Universal Robots PolyScope program: asm_idler_pulley_v1.urp

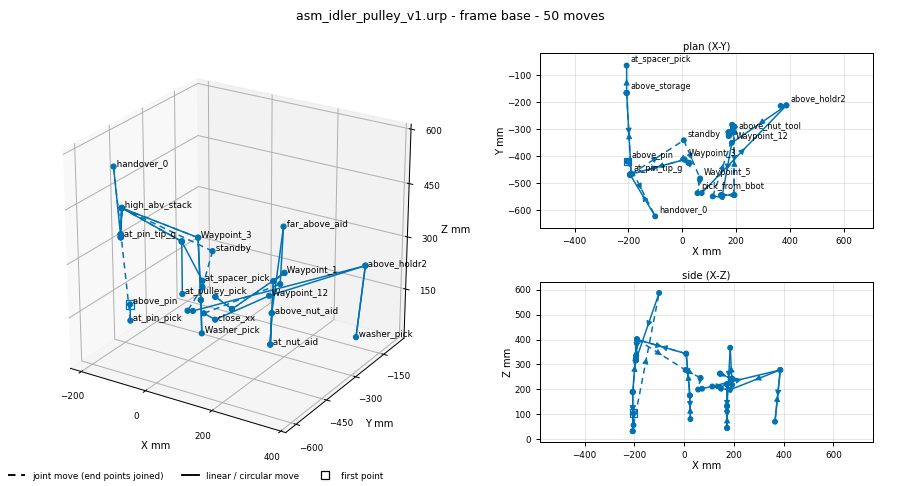
[picture p0: tool path of asm_idler_pulley_v1.urp in frame base, 50 of 58 moves have a stored position in this frame; points joined in program order, loops and branches not executed]
Program asm_idler_pulley_v1 (installation=default directory=/programs/wrs2020 createdIn=5.6.0.90886 lastSavedIn=5.9.1.1031110 robotSerialNumber=20205500180)
Calibrated DH parameters: a=[0, -0.425, -0.3922, 0, 0, 0]; d=[0.1625, 0, 0, 0.1333, 0.0997, 0.0996]; alpha=[1.570796, 0, 0, 1.570796, -1.570796, 0]; deltaTheta=[0, 0, 0, 0, 0, 0]
Robot Program (runOnlyOnce=true)
  var_1 := get_actual_joint_positions()
  MoveJ speed 60 deg/s, acceleration 80 deg/s^2 (useActiveTCP=true) feature=Base
    Waypoint Waypoint (Variable): variable=var_1
  URCap Gripper (Robotiq_Grippers, Robotiq Inc.) dataModel(position=70.98039215686275, force=100.0, speed=0.0, positionInDouble=70.98039215686275, forceInDouble=100.0, speedInDouble=0.0, slaveIds=[9], blocking=true)
  MoveL speed 50 mm/s, acceleration 1200 mm/s^2 (useActiveTCP=true) feature=Base
    Waypoint above_pin: motionParameters(jointSpeed=1.047198 jointAcceleration=1.396263 cartesianSpeed=0.5 cartesianAcceleration=1.2); TCP in base x=-203.451 y=-419.874 z=103.99 mm, rx=-2.2531 ry=-2.1572 rz=0.0025 rad; joints [48.461, -90.908, 115.612, -114.69, -91.283, 50.953] deg; TCP offset x=0 y=0 z=220 mm, rx=0 ry=0 rz=0 rad
    Waypoint at_pin_pick: motionParameters(jointSpeed=1.047198 jointAcceleration=1.396263 cartesianSpeed=0.5 cartesianAcceleration=1.2); TCP in base x=-203.465 y=-419.863 z=56.339 mm, rx=-2.2531 ry=-2.1571 rz=0.0025 rad; joints [48.46, -87.426, 120.005, -122.565, -91.284, 50.955] deg
  URCap Gripper (Robotiq_Grippers, Robotiq Inc.) dataModel(position=100.0, force=0.0, speed=0.0, positionInDouble=100.0, forceInDouble=0.0, speedInDouble=0.0, slaveIds=[9], blocking=true)
  MoveJ speed 60 deg/s, acceleration 80 deg/s^2 (useActiveTCP=true) feature=Base
    Waypoint handover_0: TCP in base x=-100.562 y=-623.369 z=587.469 mm, rx=1.5572 ry=0.0059 rz=0.0177 rad; joints [46.387, -101.66, 115.722, -195.155, -45.533, 181.192] deg
  Popup Message (haltProgram=false message=wait for b_bot to grasp pin. Press continue to release and proceed inputType=Text)
  URCap Gripper (Robotiq_Grippers, Robotiq Inc.) dataModel(position=34.90196078431372, force=100.0, speed=100.0, positionInDouble=34.90196078431372, forceInDouble=100.0, speedInDouble=100.0, slaveIds=[9], blocking=true)
  MoveL speed 250 mm/s, acceleration 1200 mm/s^2 (useActiveTCP=true) feature=Base
    MoveDirectionNode (selectedDirection=YPlus)
      Until DISTANCE (allowActions=false deceleration=3 distanceNodeType=STOP) Distance=0.08; motionParameters(blendRadius=0)
  Popup Message (haltProgram=false message=c when bbot moved down inputType=Text)
  Folder center pin
    MoveL speed 250 mm/s, acceleration 1200 mm/s^2 (useActiveTCP=true) feature=Base
      SuppressedNode
        Waypoint Waypoint_9: 
      Waypoint at_pin_tip_g: TCP in base x=-193.591 y=-468.719 z=318.204 mm, rx=3.1358 ry=0.014 rz=0.0168 rad; joints [51.873, -89.96, 82.562, -82.478, -89.318, 141.361] deg
    URCap Gripper (Robotiq_Grippers, Robotiq Inc.) dataModel(position=100.0, force=100.0, speed=100.0, positionInDouble=100.0, forceInDouble=100.0, speedInDouble=100.0, slaveIds=[9], blocking=true)
    URCap Gripper (Robotiq_Grippers, Robotiq Inc.) dataModel(position=41.96078431372549, force=100.0, speed=100.0, positionInDouble=41.96078431372549, forceInDouble=100.0, speedInDouble=100.0, slaveIds=[9], blocking=true)
    MoveL speed 800 mm/s, acceleration 1200 mm/s^2 (useActiveTCP=true) feature=Base
      Waypoint turn_left (Relative): relativeFromPosition TCP in base x=-247.487 y=-411.573 z=65.314 mm, rx=-0.0034 ry=-3.1246 rz=-0.0244 rad; joints [43.776, -86.347, 117.339, -121.073, -91.317, -46.099] deg; TCP in base x=-247.45 y=-411.548 z=65.274 mm, rx=2.2244 ry=-2.2172 rz=-0.0361 rad; joints [43.776, -86.344, 117.339, -121.066, -91.315, -136.41] deg
    URCap Gripper (Robotiq_Grippers, Robotiq Inc.) dataModel(position=100.0, force=100.0, speed=100.0, positionInDouble=100.0, forceInDouble=100.0, speedInDouble=100.0, slaveIds=[9], blocking=true)
    URCap Gripper (Robotiq_Grippers, Robotiq Inc.) dataModel(position=57.64705882352941, force=0.0, speed=0.0, positionInDouble=57.64705882352941, forceInDouble=0.0, speedInDouble=0.0, slaveIds=[9], blocking=true)
    MoveL speed 800 mm/s, acceleration 1200 mm/s^2 (useActiveTCP=true) feature=Base
      Waypoint turn_right (Relative): relativeFromPosition TCP in base x=-247.464 y=-411.551 z=65.306 mm, rx=2.2244 ry=-2.2171 rz=-0.0361 rad; joints [43.776, -86.348, 117.34, -121.068, -91.317, -136.413] deg; TCP in base x=-247.474 y=-411.554 z=65.268 mm, rx=-0.0035 ry=-3.1247 rz=-0.0244 rad; joints [43.774, -86.343, 117.34, -121.072, -91.315, -46.098] deg
    URCap Gripper (Robotiq_Grippers, Robotiq Inc.) dataModel(position=100.0, force=100.0, speed=100.0, positionInDouble=100.0, forceInDouble=100.0, speedInDouble=100.0, slaveIds=[9], blocking=true)
    URCap Gripper (Robotiq_Grippers, Robotiq Inc.) dataModel(position=0.0, force=100.0, speed=100.0, positionInDouble=0.0, forceInDouble=100.0, speedInDouble=100.0, slaveIds=[9], blocking=true)
  Folder get pulley
    MoveL speed 300 mm/s, acceleration 1200 mm/s^2 (useActiveTCP=true) feature=Base
      Waypoint above_storage: motionParameters(jointSpeed=1.047198 jointAcceleration=1.396263 cartesianSpeed=0.5 cartesianAcceleration=1.2 blendRadius=0.05); TCP in base x=-206.583 y=-165.263 z=189.567 mm, rx=3.1359 ry=0.0138 rz=0.017 rad; joints [7.844, -127.94, 126.119, -87.608, -89.601, 97.337] deg
      Waypoint at_pulley_pick: motionParameters(jointSpeed=1.047198 jointAcceleration=1.396263 cartesianSpeed=0.5 cartesianAcceleration=1.2); TCP in base x=-206.616 y=-165.272 z=31.944 mm, rx=3.1359 ry=0.0138 rz=0.0169 rad; joints [7.841, -121.393, 147.531, -115.569, -89.599, 97.336] deg
    Folder center+grasp
      URCap Gripper (Robotiq_Grippers, Robotiq Inc.) dataModel(position=100.0, force=0.0, speed=0.0, positionInDouble=100.0, forceInDouble=0.0, speedInDouble=0.0, slaveIds=[9], blocking=true)
      URCap Gripper (Robotiq_Grippers, Robotiq Inc.) dataModel(position=45.09803921568627, force=0.0, speed=0.0, positionInDouble=45.09803921568627, forceInDouble=0.0, speedInDouble=0.0, slaveIds=[9], blocking=true)
      MoveL speed 800 mm/s, acceleration 1200 mm/s^2 (useActiveTCP=true) feature=Base
        Waypoint turn_left (Relative): relativeFromPosition TCP in base x=-247.487 y=-411.573 z=65.314 mm, rx=-0.0034 ry=-3.1246 rz=-0.0244 rad; joints [43.776, -86.347, 117.339, -121.073, -91.317, -46.099] deg; TCP in base x=-247.45 y=-411.548 z=65.274 mm, rx=2.2244 ry=-2.2172 rz=-0.0361 rad; joints [43.776, -86.344, 117.339, -121.066, -91.315, -136.41] deg
      URCap Gripper (Robotiq_Grippers, Robotiq Inc.) dataModel(position=100.0, force=0.0, speed=0.0, positionInDouble=100.0, forceInDouble=0.0, speedInDouble=0.0, slaveIds=[9], blocking=true)
      URCap Gripper (Robotiq_Grippers, Robotiq Inc.) dataModel(position=57.64705882352941, force=0.0, speed=0.0, positionInDouble=57.64705882352941, forceInDouble=0.0, speedInDouble=0.0, slaveIds=[9], blocking=true)
      MoveL speed 800 mm/s, acceleration 1200 mm/s^2 (useActiveTCP=true) feature=Base
        Waypoint turn_right (Relative): relativeFromPosition TCP in base x=-247.464 y=-411.551 z=65.306 mm, rx=2.2244 ry=-2.2171 rz=-0.0361 rad; joints [43.776, -86.348, 117.34, -121.068, -91.317, -136.413] deg; TCP in base x=-247.474 y=-411.554 z=65.268 mm, rx=-0.0035 ry=-3.1247 rz=-0.0244 rad; joints [43.774, -86.343, 117.34, -121.072, -91.315, -46.098] deg
      URCap Gripper (Robotiq_Grippers, Robotiq Inc.) dataModel(position=100.0, force=0.0, speed=0.0, positionInDouble=100.0, forceInDouble=0.0, speedInDouble=0.0, slaveIds=[9], blocking=true)
  Folder stack pulley
    MoveJ speed 60 deg/s, acceleration 80 deg/s^2 (useActiveTCP=true) feature=Base
      Waypoint high_abv_stack: TCP in base x=-189.725 y=-466.715 z=400.408 mm, rx=3.1358 ry=0.0139 rz=0.0168 rad; joints [52.084, -87.731, 67.903, -70.048, -89.314, 141.575] deg
    MoveL speed 250 mm/s, acceleration 1200 mm/s^2 (useActiveTCP=true) feature=Base
      Waypoint at_tip_1: TCP in base x=-193.581 y=-468.753 z=326.241 mm, rx=3.1357 ry=0.014 rz=0.0167 rad; joints [51.875, -89.809, 81.226, -81.299, -89.316, 141.361] deg
    Folder push_down
      p_start := get_actual_tcp_pose()
      Force Frame feature=Base; selection=[0, 0, 1, 0, 0, 0]; wrench=[-5, 0, -5, 0, 0, 0]; limitsForce=[0.005, 0.15, 0.01, 1.047198, 1.047198, 1.047198]; limitsMotion=[0.1, 0.1, 0.1, 0.349066, 0.349066, 0.349066]
        MoveL speed 5 mm/s, acceleration 5 mm/s^2 (useActiveTCP=true) feature=Base
          Loop Counting (count=1) loopVariable(name=Loop_6)
            MoveDirectionNode (selectedDirection=YPlus) feature=Base
              Until DISTANCE (allowActions=false deceleration=3 distanceNodeType=STOP) Distance=0.001; motionParameters(blendRadius=0)
            MoveDirectionNode (selectedDirection=XPlus) feature=Base
              Until DISTANCE (allowActions=false deceleration=3 distanceNodeType=STOP) Distance=0.001; motionParameters(blendRadius=0)
            MoveDirectionNode (selectedDirection=YMinus) feature=Base
              Until DISTANCE (allowActions=false deceleration=3 distanceNodeType=STOP) Distance=0.001; motionParameters(blendRadius=0)
            MoveDirectionNode (selectedDirection=YMinus) feature=Base
              Until DISTANCE (allowActions=false deceleration=3 distanceNodeType=STOP) Distance=0.001; motionParameters(blendRadius=0)
            MoveDirectionNode (selectedDirection=XMinus) feature=Base
              Until DISTANCE (allowActions=false deceleration=3 distanceNodeType=STOP) Distance=0.001; motionParameters(blendRadius=0)
            MoveDirectionNode (selectedDirection=YPlus) feature=Base
              Until DISTANCE (allowActions=false deceleration=3 distanceNodeType=STOP) Distance=0.001; motionParameters(blendRadius=0)
            MoveDirectionNode (selectedDirection=YPlus) feature=Base
              Until DISTANCE (allowActions=false deceleration=3 distanceNodeType=STOP) Distance=0.001; motionParameters(blendRadius=0)
            MoveDirectionNode (selectedDirection=XMinus) feature=Base
              Until DISTANCE (allowActions=false deceleration=3 distanceNodeType=STOP) Distance=0.001; motionParameters(blendRadius=0)
            MoveDirectionNode (selectedDirection=YMinus) feature=Base
              Until DISTANCE (allowActions=false deceleration=3 distanceNodeType=STOP) Distance=0.001; motionParameters(blendRadius=0)
            MoveDirectionNode (selectedDirection=YMinus) feature=Base
              Until DISTANCE (allowActions=false deceleration=3 distanceNodeType=STOP) Distance=0.001; motionParameters(blendRadius=0)
            MoveDirectionNode (selectedDirection=XMinus) feature=Base
              Until DISTANCE (allowActions=false deceleration=3 distanceNodeType=STOP) Distance=0.001; motionParameters(blendRadius=0)
            MoveDirectionNode (selectedDirection=YPlus) feature=Base
              Until DISTANCE (allowActions=false deceleration=3 distanceNodeType=STOP) Distance=0.001; motionParameters(blendRadius=0)
        SuppressedNode
          Wait Sleep waitTime=4
      p_now := get_actual_tcp_pose()
      d := pose_dist(p_start,p_now)
      Popup Message (haltProgram=false inputType=Variable) variable=d
      If d < 0.01
        Popup Message (haltProgram=false message=fail? inputType=Text)
    URCap Gripper (Robotiq_Grippers, Robotiq Inc.) dataModel(position=41.96078431372549, force=100.0, speed=100.0, positionInDouble=41.96078431372549, forceInDouble=100.0, speedInDouble=100.0, slaveIds=[9], blocking=true)
    Folder recenter pin
      MoveL speed 250 mm/s, acceleration 1200 mm/s^2 (useActiveTCP=true) feature=Base
        Waypoint at_pin_tip_g: TCP in base x=-193.591 y=-468.719 z=318.204 mm, rx=3.1358 ry=0.014 rz=0.0168 rad; joints [51.873, -89.96, 82.562, -82.478, -89.318, 141.361] deg
      URCap Gripper (Robotiq_Grippers, Robotiq Inc.) dataModel(position=100.0, force=100.0, speed=100.0, positionInDouble=100.0, forceInDouble=100.0, speedInDouble=100.0, slaveIds=[9], blocking=true)
      URCap Gripper (Robotiq_Grippers, Robotiq Inc.) dataModel(position=41.96078431372549, force=100.0, speed=100.0, positionInDouble=41.96078431372549, forceInDouble=100.0, speedInDouble=100.0, slaveIds=[9], blocking=true)
    MoveJ speed 60 deg/s, acceleration 80 deg/s^2 (useActiveTCP=true) feature=Base
      Waypoint high_abv_stack: TCP in base x=-189.725 y=-466.715 z=400.408 mm, rx=3.1358 ry=0.0139 rz=0.0168 rad; joints [52.084, -87.731, 67.903, -70.048, -89.314, 141.575] deg
  Folder get spacer
    MoveL speed 300 mm/s, acceleration 1200 mm/s^2 (useActiveTCP=true) feature=Base
      Waypoint above_storage: motionParameters(jointSpeed=1.047198 jointAcceleration=1.396263 cartesianSpeed=0.5 cartesianAcceleration=1.2 blendRadius=0.05); TCP in base x=-206.583 y=-165.263 z=189.567 mm, rx=3.1359 ry=0.0138 rz=0.017 rad; joints [7.844, -127.94, 126.119, -87.608, -89.601, 97.337] deg
      Waypoint at_spacer_pick: motionParameters(jointSpeed=1.047198 jointAcceleration=1.396263 cartesianSpeed=0.5 cartesianAcceleration=1.2); TCP in base x=-206.636 y=-63.72 z=31.971 mm, rx=3.1359 ry=0.0138 rz=0.0168 rad; joints [-21.062, -135.483, 151.426, -105.257, -89.924, 68.434] deg
    Folder center+grasp
      URCap Gripper (Robotiq_Grippers, Robotiq Inc.) dataModel(position=100.0, force=0.0, speed=0.0, positionInDouble=100.0, forceInDouble=0.0, speedInDouble=0.0, slaveIds=[9], blocking=true)
      URCap Gripper (Robotiq_Grippers, Robotiq Inc.) dataModel(position=61.96078431372549, force=100.0, speed=0.0, positionInDouble=61.96078431372549, forceInDouble=100.0, speedInDouble=0.0, slaveIds=[9], blocking=true)
      MoveL speed 800 mm/s, acceleration 1200 mm/s^2 (useActiveTCP=true) feature=Base
        Waypoint turn_left (Relative): relativeFromPosition TCP in base x=-247.487 y=-411.573 z=65.314 mm, rx=-0.0034 ry=-3.1246 rz=-0.0244 rad; joints [43.776, -86.347, 117.339, -121.073, -91.317, -46.099] deg; TCP in base x=-247.45 y=-411.548 z=65.274 mm, rx=2.2244 ry=-2.2172 rz=-0.0361 rad; joints [43.776, -86.344, 117.339, -121.066, -91.315, -136.41] deg
      URCap Gripper (Robotiq_Grippers, Robotiq Inc.) dataModel(position=100.0, force=0.0, speed=0.0, positionInDouble=100.0, forceInDouble=0.0, speedInDouble=0.0, slaveIds=[9], blocking=true)
      URCap Gripper (Robotiq_Grippers, Robotiq Inc.) dataModel(position=57.64705882352941, force=0.0, speed=0.0, positionInDouble=57.64705882352941, forceInDouble=0.0, speedInDouble=0.0, slaveIds=[9], blocking=true)
      MoveL speed 800 mm/s, acceleration 1200 mm/s^2 (useActiveTCP=true) feature=Base
        Waypoint turn_right (Relative): relativeFromPosition TCP in base x=-247.464 y=-411.551 z=65.306 mm, rx=2.2244 ry=-2.2171 rz=-0.0361 rad; joints [43.776, -86.348, 117.34, -121.068, -91.317, -136.413] deg; TCP in base x=-247.474 y=-411.554 z=65.268 mm, rx=-0.0035 ry=-3.1247 rz=-0.0244 rad; joints [43.774, -86.343, 117.34, -121.072, -91.315, -46.098] deg
      URCap Gripper (Robotiq_Grippers, Robotiq Inc.) dataModel(position=100.0, force=0.0, speed=0.0, positionInDouble=100.0, forceInDouble=0.0, speedInDouble=0.0, slaveIds=[9], blocking=true)
    MoveL speed 300 mm/s, acceleration 1200 mm/s^2 (useActiveTCP=true) feature=Base
      Waypoint above_storage: motionParameters(jointSpeed=1.047198 jointAcceleration=1.396263 cartesianSpeed=0.5 cartesianAcceleration=1.2); TCP in base x=-206.583 y=-165.263 z=189.567 mm, rx=3.1359 ry=0.0138 rz=0.017 rad; joints [7.844, -127.94, 126.119, -87.608, -89.601, 97.337] deg
  Folder stack spacer
    MoveJ speed 60 deg/s, acceleration 80 deg/s^2 (useActiveTCP=true) feature=Base
      Waypoint high_abv_stack: TCP in base x=-189.725 y=-466.715 z=400.408 mm, rx=3.1358 ry=0.0139 rz=0.0168 rad; joints [52.084, -87.731, 67.903, -70.048, -89.314, 141.575] deg
    MoveL speed 250 mm/s, acceleration 1200 mm/s^2 (useActiveTCP=true) feature=Base
      Waypoint at_tip_1: TCP in base x=-193.581 y=-468.753 z=326.241 mm, rx=3.1357 ry=0.014 rz=0.0167 rad; joints [51.875, -89.809, 81.226, -81.299, -89.316, 141.361] deg
    Folder push_down
      p_start := get_actual_tcp_pose()
      Force Frame feature=Base; selection=[0, 0, 1, 0, 0, 0]; wrench=[-5, 0, -5, 0, 0, 0]; limitsForce=[0.005, 0.15, 0.01, 1.047198, 1.047198, 1.047198]; limitsMotion=[0.1, 0.1, 0.1, 0.349066, 0.349066, 0.349066]
        MoveL speed 5 mm/s, acceleration 5 mm/s^2 (useActiveTCP=true) feature=Base
          Loop Counting (count=1) loopVariable(name=Loop_3)
            MoveDirectionNode (selectedDirection=YPlus) feature=Base
              Until DISTANCE (allowActions=false deceleration=3 distanceNodeType=STOP) Distance=0.001; motionParameters(blendRadius=0)
            MoveDirectionNode (selectedDirection=XPlus) feature=Base
              Until DISTANCE (allowActions=false deceleration=3 distanceNodeType=STOP) Distance=0.001; motionParameters(blendRadius=0)
            MoveDirectionNode (selectedDirection=YMinus) feature=Base
              Until DISTANCE (allowActions=false deceleration=3 distanceNodeType=STOP) Distance=0.001; motionParameters(blendRadius=0)
            MoveDirectionNode (selectedDirection=YMinus) feature=Base
              Until DISTANCE (allowActions=false deceleration=3 distanceNodeType=STOP) Distance=0.001; motionParameters(blendRadius=0)
            MoveDirectionNode (selectedDirection=XMinus) feature=Base
              Until DISTANCE (allowActions=false deceleration=3 distanceNodeType=STOP) Distance=0.001; motionParameters(blendRadius=0)
            MoveDirectionNode (selectedDirection=YPlus) feature=Base
              Until DISTANCE (allowActions=false deceleration=3 distanceNodeType=STOP) Distance=0.001; motionParameters(blendRadius=0)
            MoveDirectionNode (selectedDirection=YPlus) feature=Base
              Until DISTANCE (allowActions=false deceleration=3 distanceNodeType=STOP) Distance=0.001; motionParameters(blendRadius=0)
            MoveDirectionNode (selectedDirection=XMinus) feature=Base
              Until DISTANCE (allowActions=false deceleration=3 distanceNodeType=STOP) Distance=0.001; motionParameters(blendRadius=0)
            MoveDirectionNode (selectedDirection=YMinus) feature=Base
              Until DISTANCE (allowActions=false deceleration=3 distanceNodeType=STOP) Distance=0.001; motionParameters(blendRadius=0)
            MoveDirectionNode (selectedDirection=YMinus) feature=Base
              Until DISTANCE (allowActions=false deceleration=3 distanceNodeType=STOP) Distance=0.001; motionParameters(blendRadius=0)
            MoveDirectionNode (selectedDirection=XMinus) feature=Base
              Until DISTANCE (allowActions=false deceleration=3 distanceNodeType=STOP) Distance=0.001; motionParameters(blendRadius=0)
            MoveDirectionNode (selectedDirection=YPlus) feature=Base
              Until DISTANCE (allowActions=false deceleration=3 distanceNodeType=STOP) Distance=0.001; motionParameters(blendRadius=0)
        SuppressedNode
          Wait Sleep waitTime=4
      p_now := get_actual_tcp_pose()
      d := pose_dist(p_start,p_now)
      Popup Message (haltProgram=false inputType=Variable) variable=d
      If d < 0.01
        Popup Message (haltProgram=false message=fail? inputType=Text)
    URCap Gripper (Robotiq_Grippers, Robotiq Inc.) dataModel(position=41.96078431372549, force=100.0, speed=100.0, positionInDouble=41.96078431372549, forceInDouble=100.0, speedInDouble=100.0, slaveIds=[9], blocking=true)
    Folder recenter pin
      MoveL speed 250 mm/s, acceleration 1200 mm/s^2 (useActiveTCP=true) feature=Base
        Waypoint at_pin_tip_g: TCP in base x=-193.591 y=-468.719 z=318.204 mm, rx=3.1358 ry=0.014 rz=0.0168 rad; joints [51.873, -89.96, 82.562, -82.478, -89.318, 141.361] deg
      URCap Gripper (Robotiq_Grippers, Robotiq Inc.) dataModel(position=100.0, force=100.0, speed=100.0, positionInDouble=100.0, forceInDouble=100.0, speedInDouble=100.0, slaveIds=[9], blocking=true)
      URCap Gripper (Robotiq_Grippers, Robotiq Inc.) dataModel(position=41.96078431372549, force=100.0, speed=100.0, positionInDouble=41.96078431372549, forceInDouble=100.0, speedInDouble=100.0, slaveIds=[9], blocking=true)
    MoveJ speed 60 deg/s, acceleration 80 deg/s^2 (useActiveTCP=true) feature=Base
      Waypoint high_abv_stack: TCP in base x=-189.725 y=-466.715 z=400.408 mm, rx=3.1358 ry=0.0139 rz=0.0168 rad; joints [52.084, -87.731, 67.903, -70.048, -89.314, 141.575] deg
  Folder get washer
    MoveL speed 300 mm/s, acceleration 1200 mm/s^2 (useActiveTCP=true) feature=Base
      URCap Gripper (Robotiq_Grippers, Robotiq Inc.) dataModel(position=74.50980392156863, force=100.0, speed=0.0, positionInDouble=74.50980392156863, forceInDouble=100.0, speedInDouble=0.0, slaveIds=[9], blocking=false)
      Waypoint Waypoint_3: motionParameters(blendRadius=0.05); TCP in base x=8.222 y=-412.726 z=343.306 mm, rx=3.1358 ry=0.0139 rz=0.0168 rad; joints [71.739, -102.737, 90.124, -77.5, -89.313, 161.233] deg
      Waypoint Waypoint_4: motionParameters(blendRadius=0.03); TCP in base x=22.896 y=-424.572 z=175.571 mm, rx=2.2233 ry=2.2042 rz=0.006 rad; joints [74.301, -100.95, 113.439, -102.605, -89.35, 74.795] deg
      Waypoint Washer_pick: TCP in base x=25.107 y=-424.601 z=80.478 mm, rx=2.2233 ry=2.2042 rz=0.0058 rad; joints [74.61, -95.844, 124.064, -118.346, -89.356, 75.105] deg
      URCap Gripper (Robotiq_Grippers, Robotiq Inc.) dataModel(position=100.0, force=100.0, speed=100.0, positionInDouble=100.0, forceInDouble=100.0, speedInDouble=100.0, slaveIds=[9], blocking=true)
      Waypoint Waypoint_4: motionParameters(blendRadius=0.03); TCP in base x=22.896 y=-424.572 z=175.571 mm, rx=2.2233 ry=2.2042 rz=0.006 rad; joints [74.301, -100.95, 113.439, -102.605, -89.35, 74.795] deg
      Waypoint Waypoint_3: motionParameters(blendRadius=0.05); TCP in base x=8.222 y=-412.726 z=343.306 mm, rx=3.1358 ry=0.0139 rz=0.0168 rad; joints [71.739, -102.737, 90.124, -77.5, -89.313, 161.233] deg
  Folder stack washer
    MoveJ speed 60 deg/s, acceleration 80 deg/s^2 (useActiveTCP=true) feature=Base
      Waypoint high_abv_stack: TCP in base x=-189.725 y=-466.715 z=400.408 mm, rx=3.1358 ry=0.0139 rz=0.0168 rad; joints [52.084, -87.731, 67.903, -70.048, -89.314, 141.575] deg
    MoveL speed 250 mm/s, acceleration 1200 mm/s^2 (useActiveTCP=true) feature=Base
      Waypoint at_tip_1: TCP in base x=-193.581 y=-468.753 z=326.241 mm, rx=3.1357 ry=0.014 rz=0.0167 rad; joints [51.875, -89.809, 81.226, -81.299, -89.316, 141.361] deg
    Folder push_down
      p_start := get_actual_tcp_pose()
      Force Frame feature=Base; selection=[0, 0, 1, 0, 0, 0]; wrench=[-5, 0, -5, 0, 0, 0]; limitsForce=[0.005, 0.15, 0.01, 1.047198, 1.047198, 1.047198]; limitsMotion=[0.1, 0.1, 0.1, 0.349066, 0.349066, 0.349066]
        MoveL speed 5 mm/s, acceleration 5 mm/s^2 (useActiveTCP=true) feature=Base
          Loop Counting (count=1) loopVariable(name=Loop_8)
            MoveDirectionNode (selectedDirection=YPlus) feature=Base
              Until DISTANCE (allowActions=false deceleration=3 distanceNodeType=STOP) Distance=0.001; motionParameters(blendRadius=0)
            MoveDirectionNode (selectedDirection=XPlus) feature=Base
              Until DISTANCE (allowActions=false deceleration=3 distanceNodeType=STOP) Distance=0.001; motionParameters(blendRadius=0)
            MoveDirectionNode (selectedDirection=YMinus) feature=Base
              Until DISTANCE (allowActions=false deceleration=3 distanceNodeType=STOP) Distance=0.001; motionParameters(blendRadius=0)
            MoveDirectionNode (selectedDirection=YMinus) feature=Base
              Until DISTANCE (allowActions=false deceleration=3 distanceNodeType=STOP) Distance=0.001; motionParameters(blendRadius=0)
            MoveDirectionNode (selectedDirection=XMinus) feature=Base
              Until DISTANCE (allowActions=false deceleration=3 distanceNodeType=STOP) Distance=0.001; motionParameters(blendRadius=0)
            MoveDirectionNode (selectedDirection=YPlus) feature=Base
              Until DISTANCE (allowActions=false deceleration=3 distanceNodeType=STOP) Distance=0.001; motionParameters(blendRadius=0)
            MoveDirectionNode (selectedDirection=YPlus) feature=Base
              Until DISTANCE (allowActions=false deceleration=3 distanceNodeType=STOP) Distance=0.001; motionParameters(blendRadius=0)
            MoveDirectionNode (selectedDirection=XMinus) feature=Base
              Until DISTANCE (allowActions=false deceleration=3 distanceNodeType=STOP) Distance=0.001; motionParameters(blendRadius=0)
            MoveDirectionNode (selectedDirection=YMinus) feature=Base
              Until DISTANCE (allowActions=false deceleration=3 distanceNodeType=STOP) Distance=0.001; motionParameters(blendRadius=0)
            MoveDirectionNode (selectedDirection=YMinus) feature=Base
              Until DISTANCE (allowActions=false deceleration=3 distanceNodeType=STOP) Distance=0.001; motionParameters(blendRadius=0)
            MoveDirectionNode (selectedDirection=XMinus) feature=Base
              Until DISTANCE (allowActions=false deceleration=3 distanceNodeType=STOP) Distance=0.001; motionParameters(blendRadius=0)
            MoveDirectionNode (selectedDirection=YPlus) feature=Base
              Until DISTANCE (allowActions=false deceleration=3 distanceNodeType=STOP) Distance=0.001; motionParameters(blendRadius=0)
        SuppressedNode
          Wait Sleep waitTime=4
      d := pose_dist(p_start,get_actual_tcp_pose())
      Popup Message (haltProgram=false inputType=Variable) variable=d
    URCap Gripper (Robotiq_Grippers, Robotiq Inc.) dataModel(position=41.96078431372549, force=100.0, speed=100.0, positionInDouble=41.96078431372549, forceInDouble=100.0, speedInDouble=100.0, slaveIds=[9], blocking=true)
    Folder recenter pin
      MoveL speed 250 mm/s, acceleration 1200 mm/s^2 (useActiveTCP=true) feature=Base
        Waypoint at_pin_tip_g: TCP in base x=-193.591 y=-468.719 z=318.204 mm, rx=3.1358 ry=0.014 rz=0.0168 rad; joints [51.873, -89.96, 82.562, -82.478, -89.318, 141.361] deg
      URCap Gripper (Robotiq_Grippers, Robotiq Inc.) dataModel(position=100.0, force=100.0, speed=100.0, positionInDouble=100.0, forceInDouble=100.0, speedInDouble=100.0, slaveIds=[9], blocking=true)
      URCap Gripper (Robotiq_Grippers, Robotiq Inc.) dataModel(position=41.96078431372549, force=100.0, speed=100.0, positionInDouble=41.96078431372549, forceInDouble=100.0, speedInDouble=100.0, slaveIds=[9], blocking=true)
    MoveJ speed 60 deg/s, acceleration 80 deg/s^2 (useActiveTCP=true) feature=Base
      Waypoint high_abv_stack: TCP in base x=-189.725 y=-466.715 z=400.408 mm, rx=3.1358 ry=0.0139 rz=0.0168 rad; joints [52.084, -87.731, 67.903, -70.048, -89.314, 141.575] deg
  MoveJ speed 60 deg/s, acceleration 80 deg/s^2 (useActiveTCP=true) feature=Base
    Waypoint standby: TCP in base x=5.685 y=-341.026 z=277.744 mm, rx=1.9655 ry=1.8527 rz=-0.5986 rad; joints [45.817, -147.761, 131.138, -100.105, -70.163, 53.959] deg
  Popup Message (haltProgram=false message=wait until bbot inclined stack. continue to grasp pulley inputType=Text)
  MoveJ speed 60 deg/s, acceleration 80 deg/s^2 (useActiveTCP=true) feature=Base
    Waypoint Waypoint_5: TCP in base x=65.954 y=-482.528 z=246.175 mm, rx=1.6878 ry=1.745 rz=-0.8022 rad; joints [73.284, -121.144, 142.903, -159.776, -77.596, 76.918] deg
    Waypoint pick_from_bbot: TCP in base x=56.138 y=-537.361 z=199.319 mm, rx=1.6878 ry=1.745 rz=-0.8023 rad; joints [74.647, -104.561, 142.307, -175.957, -78.611, 77.846] deg
    URCap Gripper (Robotiq_Grippers, Robotiq Inc.) dataModel(position=100.0, force=100.0, speed=0.0, positionInDouble=100.0, forceInDouble=100.0, speedInDouble=0.0, slaveIds=[9], blocking=true)
  Popup Message (haltProgram=false message=wait for bbot retreat. continue to insert into ridge inputType=Text)
  MoveL speed 10 mm/s, acceleration 50 mm/s^2 (useActiveTCP=true) feature=Base
    Waypoint hold_at_ridge: TCP in base x=71.967 y=-536.845 z=202.631 mm, rx=1.6877 ry=1.745 rz=-0.8023 rad; joints [77.866, -104.296, 141.604, -175.904, -81.017, 80.016] deg
  Popup Message (haltProgram=false message=wait for padless tool to tension. c to open slightly and wait inputType=Text)
  URCap Gripper (Robotiq_Grippers, Robotiq Inc.) dataModel(position=64.70588235294117, force=0.0, speed=0.0, positionInDouble=64.70588235294117, forceInDouble=0.0, speedInDouble=0.0, slaveIds=[9], blocking=true)
  Popup Message (haltProgram=false message=wait for tool to incline. c to move away and get washer inputType=Text)
  URCap Gripper (Robotiq_Grippers, Robotiq Inc.) dataModel(position=54.11764705882353, force=0.0, speed=0.0, positionInDouble=54.11764705882353, forceInDouble=0.0, speedInDouble=0.0, slaveIds=[9], blocking=true)
  Folder move away, get washer2
    MoveL speed 250 mm/s, acceleration 1200 mm/s^2 (useActiveTCP=true) feature=Joint_6_name
      MoveDirectionNode (selectedDirection=ZMinus)
        Until DISTANCE (allowActions=false deceleration=3 distanceNodeType=BLEND) Distance=0.15; motionParameters(blendRadius=0.05)
    MoveL speed 250 mm/s, acceleration 1200 mm/s^2 (useActiveTCP=true) feature=Base
      Waypoint above_holdr2: motionParameters(blendRadius=0.018); TCP in base x=386.166 y=-211.525 z=278.141 mm, rx=1.7275 ry=1.7878 rz=0.7731 rad; joints [95.779, -126.547, 127.795, -94.013, -44.077, 94.985] deg
      Waypoint washer_pick: TCP in base x=364.949 y=-213.418 z=70.097 mm, rx=1.8852 ry=1.8801 rz=0.5952 rad; joints [102.407, -112.29, 149.182, -134.579, -56.312, 104.892] deg
      URCap Gripper (Robotiq_Grippers, Robotiq Inc.) dataModel(position=100.0, force=100.0, speed=0.0, positionInDouble=100.0, forceInDouble=100.0, speedInDouble=0.0, slaveIds=[9], blocking=true)
      MoveDirectionNode (selectedDirection=YPlus) feature=Joint_6_name
        Until DISTANCE (allowActions=false deceleration=3 distanceNodeType=BLEND) Distance=0.05; motionParameters(blendRadius=0.02)
      Waypoint above_holdr2: motionParameters(blendRadius=0.05); TCP in base x=386.166 y=-211.525 z=278.141 mm, rx=1.7275 ry=1.7878 rz=0.7731 rad; joints [95.779, -126.547, 127.795, -94.013, -44.077, 94.985] deg
      Waypoint Waypoint_12: motionParameters(blendRadius=0.05); TCP in base x=183.744 y=-350.619 z=198.32 mm, rx=-2.2049 ry=-2.1905 rz=0.0293 rad; joints [99.672, -104.48, 112.492, -97.064, -91.986, 100.064] deg
      Waypoint close_xx: motionParameters(blendRadius=0.02); TCP in base x=147.498 y=-550.961 z=203.301 mm, rx=-2.2049 ry=-2.1905 rz=0.0294 rad; joints [92.672, -80.053, 88.445, -97.698, -92.088, 93.059] deg
      Waypoint Waypoint_8: motionParameters(jointSpeed=1.047198 jointAcceleration=1.396263 cartesianSpeed=0.05 cartesianAcceleration=1.2); TCP in base x=113.078 y=-549.296 z=211.62 mm, rx=-2.205 ry=-2.191 rz=0.0278 rad; joints [89.092, -81.595, 89.055, -96.876, -92.068, 89.468] deg
      Force Frame feature=Base; selection=[1, 0, 0, 0, 0, 0]; wrench=[-5, 0, -5, 0, 0, 0]; limitsForce=[0.005, 0.15, 0.01, 1.047198, 1.047198, 1.047198]; limitsMotion=[0.1, 0.1, 0.1, 0.349066, 0.349066, 0.349066]
        MoveL speed 5 mm/s, acceleration 10 mm/s^2 (useActiveTCP=true) feature=Base
          Loop Counting (count=1) loopVariable(name=Loop_2)
            MoveDirectionNode (selectedDirection=YPlus) feature=Base
              Until DISTANCE (allowActions=false deceleration=3 distanceNodeType=STOP) Distance=0.001; motionParameters(blendRadius=0)
            MoveDirectionNode (selectedDirection=ZPlus) feature=Base
              Until DISTANCE (allowActions=false deceleration=3 distanceNodeType=STOP) Distance=0.001; motionParameters(blendRadius=0)
            MoveDirectionNode (selectedDirection=YMinus) feature=Base
              Until DISTANCE (allowActions=false deceleration=3 distanceNodeType=STOP) Distance=0.001; motionParameters(blendRadius=0)
            MoveDirectionNode (selectedDirection=YMinus) feature=Base
              Until DISTANCE (allowActions=false deceleration=3 distanceNodeType=STOP) Distance=0.001; motionParameters(blendRadius=0)
            MoveDirectionNode (selectedDirection=ZMinus) feature=Base
              Until DISTANCE (allowActions=false deceleration=3 distanceNodeType=STOP) Distance=0.001; motionParameters(blendRadius=0)
            MoveDirectionNode (selectedDirection=YPlus) feature=Base
              Until DISTANCE (allowActions=false deceleration=3 distanceNodeType=STOP) Distance=0.001; motionParameters(blendRadius=0)
            MoveDirectionNode (selectedDirection=YPlus) feature=Base
              Until DISTANCE (allowActions=false deceleration=3 distanceNodeType=STOP) Distance=0.001; motionParameters(blendRadius=0)
            MoveDirectionNode (selectedDirection=ZMinus) feature=Base
              Until DISTANCE (allowActions=false deceleration=3 distanceNodeType=STOP) Distance=0.001; motionParameters(blendRadius=0)
            MoveDirectionNode (selectedDirection=YMinus) feature=Base
              Until DISTANCE (allowActions=false deceleration=3 distanceNodeType=STOP) Distance=0.001; motionParameters(blendRadius=0)
            MoveDirectionNode (selectedDirection=YMinus) feature=Base
              Until DISTANCE (allowActions=false deceleration=3 distanceNodeType=STOP) Distance=0.001; motionParameters(blendRadius=0)
            MoveDirectionNode (selectedDirection=ZMinus) feature=Base
              Until DISTANCE (allowActions=false deceleration=3 distanceNodeType=STOP) Distance=0.001; motionParameters(blendRadius=0)
            MoveDirectionNode (selectedDirection=YPlus) feature=Base
              Until DISTANCE (allowActions=false deceleration=3 distanceNodeType=STOP) Distance=0.001; motionParameters(blendRadius=0)
        SuppressedNode
          Wait Sleep waitTime=4
      URCap Gripper (Robotiq_Grippers, Robotiq Inc.) dataModel(position=60.3921568627451, force=100.0, speed=0.0, positionInDouble=60.3921568627451, forceInDouble=100.0, speedInDouble=0.0, slaveIds=[9], blocking=true)
      MoveDirectionNode (selectedDirection=XPlus)
        Until DISTANCE (allowActions=false deceleration=3 distanceNodeType=STOP) Distance=0.05; motionParameters(blendRadius=0)
    MoveJ speed 60 deg/s, acceleration 80 deg/s^2 (useActiveTCP=true) feature=Base
      Waypoint above_nut_tool: TCP in base x=192.885 y=-311.331 z=218.062 mm, rx=3.1313 ry=0.0035 rz=0.0125 rad; joints [100.109, -111.334, 114.534, -93.861, -89.651, 189.982] deg
  Popup Message (haltProgram=false message=call nut routine inputType=Text)
  Folder nut routine
    MoveL speed 250 mm/s, acceleration 1200 mm/s^2 (useActiveTCP=true) feature=Base
      Waypoint far_above_aid: TCP in base x=185.019 y=-283.793 z=367.304 mm, rx=3.0427 ry=0.0266 rz=0.0843 rad; joints [97.518, -117.381, 97.301, -75.775, -87.414, -173.456] deg
    MoveL speed 250 mm/s, acceleration 1200 mm/s^2 (useActiveTCP=true) feature=Base
      Waypoint above_nut_aid: TCP in base x=172.519 y=-318.273 z=132.878 mm, rx=3.1334 ry=-0.0123 rz=-0.0179 rad; joints [97.626, -109.17, 125.745, -106.863, -90.541, -171.937] deg
      URCap Gripper (Robotiq_Grippers, Robotiq Inc.) dataModel(position=21.96078431372549, force=100.0, speed=100.0, positionInDouble=21.96078431372549, forceInDouble=100.0, speedInDouble=100.0, slaveIds=[9], blocking=true)
      Waypoint at_nut_aid: TCP in base x=172.519 y=-325.105 z=44.86 mm, rx=3.1334 ry=-0.0123 rz=-0.0179 rad; joints [97.451, -101.585, 134.781, -123.486, -90.53, -172.054] deg
      URCap Gripper (Robotiq_Grippers, Robotiq Inc.) dataModel(position=100.0, force=100.0, speed=100.0, positionInDouble=100.0, forceInDouble=100.0, speedInDouble=100.0, slaveIds=[9], blocking=true)
      Waypoint slightly_above: TCP in base x=172.519 y=-311.073 z=221.087 mm, rx=3.1334 ry=-0.0123 rz=-0.0179 rad; joints [97.806, -112.461, 114.667, -92.492, -90.559, -171.799] deg
    MoveJ speed 60 deg/s, acceleration 80 deg/s^2 (useActiveTCP=true) feature=Base
      Waypoint Waypoint_1: TCP in base x=193.098 y=-290.824 z=241.653 mm, rx=-2.26 ry=-2.0992 rz=0.0999 rad; joints [105.872, -111.142, 110.658, -88.291, -94.599, -249.911] deg
      Waypoint Waypoint_2: motionParameters(blendRadius=0.036); TCP in base x=193.098 y=-544.308 z=241.653 mm, rx=-2.26 ry=-2.0992 rz=0.0999 rad; joints [98.952, -79.277, 82.032, -92.106, -94.688, -256.794] deg
      Waypoint before_shaft: TCP in base x=144.251 y=-544.485 z=263.341 mm, rx=2.2425 ry=2.1895 rz=-0.0817 rad; joints [92.3, -83.868, 84.821, -93.226, -91.975, -266.37] deg
    MoveL speed 5 mm/s, acceleration 100 mm/s^2 (useActiveTCP=true) feature=Base
      Waypoint at_shaft (Relative): relativeFromPosition TCP in base x=144.251 y=-544.503 z=263.351 mm, rx=2.2425 ry=2.1895 rz=-0.0818 rad; joints [92.3, -83.867, 84.819, -93.228, -91.976, -266.371] deg; TCP in base x=137.728 y=-544.491 z=263.397 mm, rx=2.2425 ry=2.1895 rz=-0.0819 rad; joints [91.604, -84.12, 85.101, -93.283, -91.949, -267.066] deg
      Popup Message (haltProgram=false message=turn on motor, then press enter to start spiral motion inputType=Text)
      Force Frame feature=Base; selection=[1, 0, 0, 0, 0, 0]; wrench=[-5, 0, 10, 0, 0, 0]; limitsForce=[0.005, 0.15, 0.01, 1.047198, 1.047198, 1.047198]; limitsMotion=[0.1, 0.1, 0.1, 0.349066, 0.349066, 0.349066]
        Loop Counting (count=5) loopVariable(name=Loop_1)
          MoveDirectionNode (selectedDirection=YPlus) feature=Base
            Until DISTANCE (allowActions=false deceleration=3 distanceNodeType=STOP) Distance=0.002; motionParameters(blendRadius=0)
          MoveDirectionNode (selectedDirection=ZPlus) feature=Base
            Until DISTANCE (allowActions=false deceleration=3 distanceNodeType=STOP) Distance=0.002; motionParameters(blendRadius=0)
          MoveDirectionNode (selectedDirection=YMinus) feature=Base
            Until DISTANCE (allowActions=false deceleration=3 distanceNodeType=STOP) Distance=0.002; motionParameters(blendRadius=0)
          MoveDirectionNode (selectedDirection=YMinus) feature=Base
            Until DISTANCE (allowActions=false deceleration=3 distanceNodeType=STOP) Distance=0.002; motionParameters(blendRadius=0)
          MoveDirectionNode (selectedDirection=ZMinus) feature=Base
            Until DISTANCE (allowActions=false deceleration=3 distanceNodeType=STOP) Distance=0.002; motionParameters(blendRadius=0)
          MoveDirectionNode (selectedDirection=YPlus) feature=Base
            Until DISTANCE (allowActions=false deceleration=3 distanceNodeType=STOP) Distance=0.002; motionParameters(blendRadius=0)
          MoveDirectionNode (selectedDirection=YPlus) feature=Base
            Until DISTANCE (allowActions=false deceleration=3 distanceNodeType=STOP) Distance=0.002; motionParameters(blendRadius=0)
          MoveDirectionNode (selectedDirection=ZMinus) feature=Base
            Until DISTANCE (allowActions=false deceleration=3 distanceNodeType=STOP) Distance=0.002; motionParameters(blendRadius=0)
          MoveDirectionNode (selectedDirection=YMinus) feature=Base
            Until DISTANCE (allowActions=false deceleration=3 distanceNodeType=STOP) Distance=0.002; motionParameters(blendRadius=0)
          MoveDirectionNode (selectedDirection=YMinus) feature=Base
            Until DISTANCE (allowActions=false deceleration=3 distanceNodeType=STOP) Distance=0.002; motionParameters(blendRadius=0)
          MoveDirectionNode (selectedDirection=ZPlus) feature=Base
            Until DISTANCE (allowActions=false deceleration=3 distanceNodeType=STOP) Distance=0.002; motionParameters(blendRadius=0)
          MoveDirectionNode (selectedDirection=YPlus) feature=Base
            Until DISTANCE (allowActions=false deceleration=3 distanceNodeType=STOP) Distance=0.002; motionParameters(blendRadius=0)
    Popup Message (haltProgram=false message=ok? inputType=Text)
    MoveJ speed 60 deg/s, acceleration 80 deg/s^2 (useActiveTCP=true) feature=Base
      Waypoint before_shaft: motionParameters(jointSpeed=1.047198 jointAcceleration=1.396263 cartesianSpeed=0.25 cartesianAcceleration=1.2); TCP in base x=144.251 y=-544.485 z=263.341 mm, rx=2.2425 ry=2.1895 rz=-0.0817 rad; joints [92.3, -83.868, 84.821, -93.226, -91.975, -266.37] deg
      Waypoint Waypoint_2: motionParameters(jointSpeed=2.094395 jointAcceleration=2.094395 cartesianSpeed=0.25 cartesianAcceleration=1.2 blendRadius=0.05); TCP in base x=193.098 y=-544.308 z=241.653 mm, rx=-2.26 ry=-2.0992 rz=0.0999 rad; joints [98.952, -79.277, 82.032, -92.106, -94.688, -256.794] deg
      Waypoint Waypoint_1: motionParameters(jointSpeed=2.094395 jointAcceleration=2.094395 cartesianSpeed=0.25 cartesianAcceleration=1.2); TCP in base x=193.098 y=-290.824 z=241.653 mm, rx=-2.26 ry=-2.0992 rz=0.0999 rad; joints [105.872, -111.142, 110.658, -88.291, -94.599, -249.911] deg
    MoveL speed 250 mm/s, acceleration 1200 mm/s^2 (useActiveTCP=true) feature=Base
      Waypoint slightly_above: TCP in base x=172.519 y=-311.073 z=221.087 mm, rx=3.1334 ry=-0.0123 rz=-0.0179 rad; joints [97.806, -112.461, 114.667, -92.492, -90.559, -171.799] deg
      Waypoint at_nut_aid: TCP in base x=172.519 y=-325.105 z=44.86 mm, rx=3.1334 ry=-0.0123 rz=-0.0179 rad; joints [97.451, -101.585, 134.781, -123.486, -90.53, -172.054] deg
      URCap Gripper (Robotiq_Grippers, Robotiq Inc.) dataModel(position=21.96078431372549, force=100.0, speed=100.0, positionInDouble=21.96078431372549, forceInDouble=100.0, speedInDouble=100.0, slaveIds=[9], blocking=true)
      Waypoint above_nut_aid: TCP in base x=172.519 y=-318.273 z=132.878 mm, rx=3.1334 ry=-0.0123 rz=-0.0179 rad; joints [97.626, -109.17, 125.745, -106.863, -90.541, -171.937] deg
